// TIA Portal V18 export
DATA_BLOCK "PLC8_CPU1214_DI_Vars"   // DB11013
{ S7_Optimized_Access := 'FALSE' }
VERSION : 0.1
// stored: AutoNumber false, DBAccessibleFromOPCUA true, IsOnlyStoredInLoadMemory false, IsWriteProtectedInAS false
   VAR
      DI1 : "UDT_DIadv";   // AHU F Гот. роб. обігр. пов. засл. (1.202)
      DI2 : "UDT_DIadv";   // AHU F Термостат загр. замерз. (1.50)
      DI3 : "UDT_DIadv";   // AHU NF Авто. режим пр. вент. (1.200)
      DI4 : "UDT_DIadv";   // AHU F 1-шв. пр. вент. (1.200)
      DI5 : "UDT_DIadv";   // AHU F 2-шв. пр. вент. (1.200)
      DI6 : "UDT_DIadv";   // AHU F Тепл. реле. 1-шв. пр. вент. (1.200)
      DI7 { S7_SetPoint := 'True'} : "UDT_DIadv";   // AHU F Тепл. реле. 2-шв. пр. вент. (1.200)
      DI8 { S7_SetPoint := 'True'} : "UDT_DIadv";   // AHU F Перегрів пр. вент. (1.200)
      DI9 { S7_SetPoint := 'True'} : "UDT_DIadv";   // AHU F Інд. сервісний вимикач. пр. вент. (1.200)
      DI10 { S7_SetPoint := 'True'} : "UDT_DIadv";   // AHU F Несправність клиновий ремінь пр. вент. (1.54)
      DI11 { S7_SetPoint := 'True'} : "UDT_DIadv";   // AHU F Забруднення пр. фільтру (1.53)
      DI12 { S7_SetPoint := 'True'} : "UDT_DIadv";   // AHU F Робота цирк. насос (1.201)
      DI13 { S7_SetPoint := 'True'} : "UDT_DIadv";   // AHU F Авто режим цирк. насос (1.201)
      DI14 { S7_SetPoint := 'True'} : "UDT_DIadv";   // AHU F Перегрів цирк. насос (1.201)
   END_VAR
BEGIN
   DI1.cFuncSystemID := 3;
   DI1.cFuncVar := 19;
   DI2.cFuncSystemID := 3;
   DI2.cFuncVar := 8;
   DI3.cFuncSystemID := 3;
   DI3.cFuncVar := 9;
   DI4.cFuncSystemID := 3;
   DI4.cFuncVar := 20;
   DI5.cFuncSystemID := 3;
   DI5.cFuncVar := 7;
   DI6.cFuncSystemID := 3;
   DI6.cFuncVar := 21;
   DI8.cFuncSystemID := 10;
   DI8.cFuncVar := 41;
   DI9.cFuncSystemID := 10;
   DI9.cFuncVar := 43;
   DI10.cFuncSystemID := 3;
   DI10.cFuncVar := 16;
   DI11.cFuncSystemID := 0;
   DI11.cFuncVar := 0;
   DI12.cFuncSystemID := 0;
   DI12.cFuncVar := 0;
   DI13.cFuncSystemID := 0;
   DI13.cFuncVar := 0;
END_DATA_BLOCK
